{attribute 'qualified_only'}
VAR_GLOBAL
		//0 - Production Mode, 1 - Manual Mode, 2 - Maintenance Mode
		MenuToDisplay :INT;
		//0 - will keep MainMenu open, 1- InfoMenu overlay during the production
		PopupToDisplay :INT;		
END_VAR

(* stored: Version 1.1.0.1, ProductVersion 3.1.4024.15
   GVL GVL_HMI: Id {3f4f1fbc-c983-49da-9610-9708250e48c1} *)
